FUNCTION_BLOCK FB_SaMElementExecute EXTENDS FB_SaMElement
VAR
END_VAR

METHOD FB_init : BOOL
VAR_INPUT
	bInitRetains : BOOL; // if TRUE, the retain variables are initialized (warm start / cold start)
	bInCopyCode : BOOL;  // if TRUE, the instance afterwards gets moved into the copy code (online change)
END_VAR
THIS^.SetText (eLocation := E_BaseLocation.pl, wsDescription := "Wykonywany");
THIS^.SetText (eLocation := E_BaseLocation.en, wsDescription := "Ausführen");
THIS^.SetText (eLocation := E_BaseLocation.de, wsDescription := "Execute");
THIS^.SetName (stName := THIS^.GetTexts ());
END_METHOD

METHOD PUBLIC InvokeStateForTopElement : BOOL
VAR_INPUT
	itfTopElement		: ITF_BaseSaMStateMethod;
END_VAR
InvokeStateForTopElement	:= itfTopElement.SP_Execute ();
END_METHOD

END_FUNCTION_BLOCK

(* stored: Version 1.1.0.1
   POU FB_SaMElementExecute: Id {0330597f-6b08-0848-19eb-823cfbcb02c4}, SpecialFunc None
   Method FB_init: Id {c81d05fa-cb63-0a62-07ed-5201a5c29577}
   Method InvokeStateForTopElement: Id {82079831-919e-05ff-05ad-3973fe4d5d98} *)
